FUNCTION_BLOCK FB_NOTT_CRYO_COOLDOWN
VAR_INPUT
	in_bEnable:		BOOL := FALSE;	// System active while in_bEnable is TRUE
	in_Cryo_Stat:	T_NOTT_CRYO_STAT;
END_VAR
VAR_OUTPUT
	out_bPermit_Evacuation_Stop:	BOOL := FALSE;
	out_bPermit_WarmUp:				BOOL := FALSE;

END_VAR

VAR_IN_OUT
	{attribute 'OPC.UA.DA' := '0'}
	nott_temps:						FB_NOTT_TEMPERATURES;
	{attribute 'OPC.UA.DA' := '0'}
	nott_heaters:					FB_NOTT_HEATERS;
	{attribute 'OPC.UA.DA' := '0'}
	nott_t_ctrls:      				FB_NOTT_TCTRLs;
	{attribute 'OPC.UA.DA' := '0'}
	nott_t_votes: 					FB_NOTT_VOTERS;
END_VAR
VAR
	
	{attribute 'TcHmiSymbol.Show'}	
	cfg:	T_NOTT_CRYO_COOLDOWN_CFG;
	{attribute 'TcHmiSymbol.Show'}
	ctrl:	T_NOTT_CRYO_COOLDOWN_CTRL;

	{attribute 'OPC.UA.DA' := '1'}
	{attribute 'OPC.UA.DA.Access' := '1'}
	{attribute 'TcHmiSymbol.Show'}
	stat:	T_NOTT_CRYO_COOLDOWN_STAT;

// Cooler	
	
	{attribute 'TcHmiSymbol.Show'}
	cooler:			FB_METIS_CRYO_CPA;
	
//
// Internals
//
	timer:	TON;
	trig:	R_TRIG;	// Start trigger
//

	{attribute 'TcHmiSymbol.Show'}
	bPermitStart:	BOOL := FALSE;
	{attribute 'TcHmiSymbol.Show'}
	bPermitStop:	BOOL := FALSE;
	
END_VAR

M_Configure();
M_ExecuteControllers();
M_SafetyCheck();
M_StateMachine( 
	nott_temps  := nott_temps,
	nott_heaters := nott_heaters,
	nott_t_ctrls := nott_t_ctrls,
	nott_t_votes := nott_t_votes
);
M_UpdateStatus();

METHOD M_Configure
VAR_INPUT
END_VAR
VAR
	refBOOL:	REFERENCE TO BOOL;
END_VAR
// IF stat.bConfigured THEN
// 
// ELSE
// 	RETURN;
// END_IF
END_METHOD

METHOD M_ExecuteControllers
VAR
	ptrSimTemp:	POINTER TO LREAL;
END_VAR


	
// Hardware-level cooling veto. This prevents a stale command or scan-order
// delay from enabling the cooler before confirmed vacuum is available.
ctrl.cor_Cooler(
    in_bEnable := ctrl.bEnable_Cooler
        AND in_Cryo_Stat.bPressureValid
        AND in_Cryo_Stat.bVacuum
        AND (
            (in_Cryo_Stat.bIsPVPRunning
             AND in_Cryo_Stat.bIsTMPRunning)
            OR in_Cryo_Stat.bOP
        ));
Cooler(
	in_bEnable:= ctrl.cor_Cooler.out_bEnable,
	in_bSimulation:= FALSE, 
	in_sName:= 'PTC Cooler', 
	in_sSN_Compressor:= 'CPA28H5W2DNCE-410730000001', 
	in_sSN_PulseTube:= 'PT810-19880200001', 
	in_nYear_Compressor:= 2023, 
	in_nYear_PulseTube:= 2023, 
	in_lrNextService_Compressor:= 20000.0, 
	in_lrNextService_PulseTube:= 40000.0, 
	in_nSlaveID:= 16, 
	in_nPeriod:= 1000);
END_METHOD

METHOD M_PermitStart_Cooldown
VAR_INPUT
	in_bPermissionStart: BOOL;
END_VAR
bPermitStart := in_bPermissionStart;
END_METHOD

METHOD M_PermitStop_Cooldown
VAR_INPUT
	in_bPermissionStop: BOOL;
END_VAR
bPermitStop := in_bPermissionStop;
END_METHOD

METHOD M_SafetyCheck
VAR_INPUT
END_VAR
VAR CONSTANT
	lrPress_ColdAlarmTrip:	LREAL := 10.0E-1;	// [mbar]
	lrPress_ColdAlarmReset:	LREAL := 8.0E-1;	// [mbar], hysteresis reset
END_VAR
// Keep pressure and pump alarm causes separate so clearing one condition
// cannot hide the other.
IF NOT in_Cryo_Stat.bCold THEN
	stat.bPressureAlarm := FALSE;
ELSIF in_Cryo_Stat.bPressureValid THEN
	IF stat.bPressureAlarm THEN
		IF in_Cryo_Stat.lrPressure_mbar < lrPress_ColdAlarmReset THEN
			stat.bPressureAlarm := FALSE;
		END_IF
	ELSIF in_Cryo_Stat.lrPressure_mbar > lrPress_ColdAlarmTrip THEN
		stat.bPressureAlarm := TRUE;
	END_IF
END_IF

// A pump loss during active cooldown trips the routine. The alarm resets only
// after both pumps recover; a new operator command is required to restart.
IF stat.bActive
    AND NOT in_Cryo_Stat.bOP
    AND (NOT in_Cryo_Stat.bIsPVPRunning
         OR NOT in_Cryo_Stat.bIsTMPRunning) THEN

    stat.bPumpAlarm := TRUE;
    ctrl.bEnable_Cooler := FALSE;
    stat.nState := E_NOTT_CRYO_COOLDOWN_STATE.STOP_COOLDOWN;
    stat.sErrorText := 'Pump stopped during cooldown.';

ELSIF (in_Cryo_Stat.bIsPVPRunning
       AND in_Cryo_Stat.bIsTMPRunning)
      OR in_Cryo_Stat.bOP THEN

    stat.bPumpAlarm := FALSE;
END_IF


stat.bAlarm := stat.bPressureAlarm OR stat.bPumpAlarm;
stat.bWarning := stat.bAlarm;
END_METHOD

METHOD M_StateMachine : BOOL
VAR_INPUT
END_VAR
VAR_IN_OUT
	{attribute 'OPC.UA.DA' := '0'}
	nott_temps:						FB_NOTT_TEMPERATURES;
	{attribute 'OPC.UA.DA' := '0'}
	nott_heaters:					FB_NOTT_HEATERS;
	{attribute 'OPC.UA.DA' := '0'}
	nott_t_ctrls:      				FB_NOTT_TCTRLs;
	{attribute 'OPC.UA.DA' := '0'}
	nott_t_votes: 					FB_NOTT_VOTERS;
END_VAR
VAR_INST
    tonStopCooldown : TON;
END_VAR
M_StateMachine := FALSE;

// The routine cannot remain in a cooling state without confirmed vacuum.
// The actuator is already vetoed in M_ExecuteControllers(); this transition
// keeps the routine state and HMI status consistent with physical safety.
IF ((stat.nState = E_NOTT_CRYO_COOLDOWN_STATE.START_PTC)
	OR (stat.nState = E_NOTT_CRYO_COOLDOWN_STATE.START_RAMPDOWN_DETECTOR)
	OR (stat.nState = E_NOTT_CRYO_COOLDOWN_STATE.COOLING)
	OR (stat.nState = E_NOTT_CRYO_COOLDOWN_STATE.OPERATIONAL_TEMPERATURE_ACHIEVED))
	AND (NOT in_Cryo_Stat.bPressureValid OR NOT in_Cryo_Stat.bVacuum) THEN
	ctrl.bEnable_Cooler := FALSE;
	stat.nState := E_NOTT_CRYO_COOLDOWN_STATE.STOP_COOLDOWN;
	stat.sStatus := 'Stopping cooldown: vacuum lost or pressure invalid.';
END_IF

CASE stat.nState OF

    E_NOTT_CRYO_COOLDOWN_STATE.NONE:
        // Nothing to do here
        stat.sStatus := 'NONE';
		stat.bActive := FALSE;
		stat.nState := E_NOTT_CRYO_COOLDOWN_STATE.OFF;

    E_NOTT_CRYO_COOLDOWN_STATE.OFF:

        ctrl.cor_Cooler.M_SetPermissions(FALSE, TRUE); // Only OFF allowed

        stat.sState  := 'OFF';
        stat.sStatus := 'OFF';

        ctrl.bEnable_Cooler := FALSE;

        out_bPermit_Evacuation_Stop := TRUE;
        out_bPermit_WarmUp          := TRUE;
		stat.bActive := FALSE;
		
        trig(CLK := in_bEnable);

        IF trig.Q
		   AND in_Cryo_Stat.bPressureValid
		   AND in_Cryo_Stat.bVacuum
		   AND in_Cryo_Stat.bIsPVPRunning
		   AND in_Cryo_Stat.bIsTMPRunning THEN
            stat.nState := E_NOTT_CRYO_COOLDOWN_STATE.START_PTC;
            stat.sStatus := 'Starting PTC...';

            out_bPermit_Evacuation_Stop := FALSE;
            out_bPermit_WarmUp          := FALSE;
			
			stat.bActive := TRUE;
		ELSIF trig.Q THEN
			stat.sStatus := 'Cooldown start rejected: vacuum/pumps not ready.';
        END_IF;


    E_NOTT_CRYO_COOLDOWN_STATE.START_PTC:
		stat.bActive := TRUE;
		ctrl.cor_Cooler.M_SetPermissions(TRUE, TRUE);

		out_bPermit_Evacuation_Stop := FALSE;
		out_bPermit_WarmUp          := FALSE;

		IF NOT in_bEnable THEN
			ctrl.bEnable_Cooler := FALSE;
			stat.nState := E_NOTT_CRYO_COOLDOWN_STATE.STOP_COOLDOWN;
			stat.sStatus := 'Cooldown cancelled while starting PTC...';
		ELSE
			ctrl.bEnable_Cooler := TRUE;

			IF cooler.stat.bSystemOn THEN
				stat.nState := E_NOTT_CRYO_COOLDOWN_STATE.START_RAMPDOWN_DETECTOR;
				stat.sStatus := 'PTC started. Starting detector ramp down...';
			END_IF
		END_IF


    E_NOTT_CRYO_COOLDOWN_STATE.START_RAMPDOWN_DETECTOR:
		ctrl.cor_Cooler.M_SetPermissions(TRUE, TRUE);
		ctrl.bEnable_Cooler := TRUE;

		IF NOT in_bEnable THEN
			ctrl.bEnable_Cooler := FALSE;
			stat.nState := E_NOTT_CRYO_COOLDOWN_STATE.STOP_COOLDOWN;
			stat.sStatus := 'Stopping cooldown...';
			RETURN;
		END_IF

        // Enable detector heaters
        nott_heaters.h_detector.M_SetEnable();
        nott_heaters.h_detector_spare.M_SetEnable();

        // Enable detector temperature control loops
        nott_t_ctrls.tc_detector.M_SetEnable();
        nott_t_ctrls.tc_detector_spare.M_SetEnable();

        // Set detector setpoints
        nott_t_ctrls.tc_detector.M_Set_SetPoint(
            m_eSetpointType    := E_METIS_CTRL_SETPOINT_SWITCH.FIXED,
            m_lrFixedSetpoint  := cfg.lrTemp_Det,
            m_lrSetpointOffset := 0.0,
            m_pSetpointTemp    := nott_temps.M_SetTemperatureSensor(0)
        );

        nott_t_ctrls.tc_detector_spare.M_Set_SetPoint(
            m_eSetpointType    := E_METIS_CTRL_SETPOINT_SWITCH.FIXED,
            m_lrFixedSetpoint  := cfg.lrTemp_Det,
            m_lrSetpointOffset := 0.0,
            m_pSetpointTemp    := nott_temps.M_SetTemperatureSensor(0)
        );

        stat.sStatus := 'Detector ramp down active...';

        stat.nState := E_NOTT_CRYO_COOLDOWN_STATE.COOLING;
		stat.bActive := TRUE;

    E_NOTT_CRYO_COOLDOWN_STATE.COOLING:
		ctrl.cor_Cooler.M_SetPermissions(TRUE, TRUE);
		ctrl.bEnable_Cooler := TRUE;

        out_bPermit_Evacuation_Stop := FALSE;
        out_bPermit_WarmUp          := FALSE;
		stat.bActive := TRUE;
        IF in_bEnable THEN

            IF in_Cryo_Stat.bOP THEN

                stat.sStatus := 'Operational temperature achieved.';
                stat.nState  := E_NOTT_CRYO_COOLDOWN_STATE.OPERATIONAL_TEMPERATURE_ACHIEVED;

            ELSE
                stat.sStatus := 'Cooling...';
            END_IF;

        ELSE
            stat.nState := E_NOTT_CRYO_COOLDOWN_STATE.STOP_COOLDOWN;
            stat.sStatus := 'Stopping cooldown...';
        END_IF;


    E_NOTT_CRYO_COOLDOWN_STATE.OPERATIONAL_TEMPERATURE_ACHIEVED:
		stat.bActive := TRUE;
		ctrl.cor_Cooler.M_SetPermissions(TRUE, TRUE);
		ctrl.bEnable_Cooler := TRUE;
        IF in_bEnable THEN
			IF NOT in_Cryo_Stat.bOP THEN
				out_bPermit_Evacuation_Stop := FALSE;
				out_bPermit_WarmUp          := FALSE;
				stat.nState := E_NOTT_CRYO_COOLDOWN_STATE.COOLING;
				stat.sStatus := 'Operational state lost. Resuming cooldown...';
			ELSE
                stat.sStatus := 'Operational temperature achieved.';

                out_bPermit_Evacuation_Stop := TRUE;
                out_bPermit_WarmUp          := FALSE;
			END_IF

        ELSE
            stat.nState := E_NOTT_CRYO_COOLDOWN_STATE.STOP_COOLDOWN;
            stat.sStatus := 'Stopping cooldown...';

            out_bPermit_Evacuation_Stop := FALSE;
            out_bPermit_WarmUp          := FALSE;
        END_IF;


    E_NOTT_CRYO_COOLDOWN_STATE.STOP_COOLDOWN:
		stat.bActive := TRUE;
		// Disable PTC
		ctrl.cor_Cooler.M_SetPermissions(FALSE, TRUE);
		ctrl.bEnable_Cooler := FALSE;
	
		out_bPermit_Evacuation_Stop := FALSE;
		out_bPermit_WarmUp          := FALSE;
	
		// Keep detector protection active
		nott_heaters.h_detector.M_SetEnable();
		nott_heaters.h_detector_spare.M_SetEnable();
	
		nott_t_ctrls.tc_detector.M_SetEnable();
		nott_t_ctrls.tc_detector_spare.M_SetEnable();
	
		// Follow the lowest cryostat temperature +10 K
		nott_t_ctrls.tc_detector.M_Set_SetPoint(
			m_eSetpointType    := E_METIS_CTRL_SETPOINT_SWITCH.FIXED,
			m_lrFixedSetpoint  := nott_temps.out_lrLowestTemp,
			m_lrSetpointOffset := 10.0,
			m_pSetpointTemp    := nott_temps.M_SetTemperatureSensor(0));
	
		nott_t_ctrls.tc_detector_spare.M_Set_SetPoint(
			m_eSetpointType    := E_METIS_CTRL_SETPOINT_SWITCH.FIXED,
			m_lrFixedSetpoint  := nott_temps.out_lrLowestTemp,
			m_lrSetpointOffset := 10.0,
			m_pSetpointTemp    := nott_temps.M_SetTemperatureSensor(0));
	
		stat.sStatus := 'Waiting for detector protection...';
	
		// Safety timeout (e.g. 5 minutes)
		tonStopCooldown(IN := TRUE, PT := T#15M);
	
		IF ((nott_t_votes.vote_detector.stat.bValid
			AND nott_temps.out_bLowestTempValid
			AND (nott_t_votes.vote_detector.stat.lrTempK >= (nott_temps.out_lrLowestTemp + 8.0)))
			OR tonStopCooldown.Q) THEN
	
			tonStopCooldown(IN := FALSE);
	
			stat.sStatus := 'Cooldown stopped.';
			stat.nState := E_NOTT_CRYO_COOLDOWN_STATE.OFF;
			stat.bActive := FALSE;
		END_IF;


ELSE
    stat.nState  := E_NOTT_CRYO_COOLDOWN_STATE.NONE;
    stat.sStatus := 'UNKNOWN STATE';
	stat.bActive := FALSE;
END_CASE;

M_StateMachine := TRUE;
END_METHOD

METHOD M_UpdateStatus : BOOL
VAR_INPUT
END_VAR
stat.bEnabled		:= in_bEnable;
END_METHOD

END_FUNCTION_BLOCK

(* stored: Version 1.1.0.1, ProductVersion 3.1.4026.18
   POU FB_NOTT_CRYO_COOLDOWN: Id {3d276ebb-7af3-413c-9feb-e00a6a8d77c1}, SpecialFunc None
   Method M_Configure: Id {ccc9267f-822f-4685-96df-ac997867417a}
   Method M_ExecuteControllers: Id {8cc20e87-b626-4c5a-9321-01e3b09d7bff}
   Method M_PermitStart_Cooldown: Id {95df11b7-4bb9-482f-b138-99b0dcae3606}
   Method M_PermitStop_Cooldown: Id {be3e58f2-d762-45b8-8be2-732b8074256e}
   Method M_SafetyCheck: Id {5c029b7a-7ff4-42d5-b9d2-5d6029555fd7}
   Method M_StateMachine: Id {7abd98e3-84d4-4188-bcad-d6dcca952a4b}
   Method M_UpdateStatus: Id {322aef71-4cd7-4e8d-8c64-bfe31c78f2b3} *)
